PROGRAM MAIN
VAR
	linear_phy_to_adc_test_ 		: linear_phy_to_adc_test;
	linear_adc_to_phy_test_ 		: linear_adc_to_phy_test;
	InterfaceManager_test_ 			: InterfaceManager_test;
	
	coe_handler : CoE_communication_handler;
	interface_manager :InterfaceManager;

	// Terminal_1 : EK1101
	Terminal_2 : EL1808(CoE_communication_handler:=coe_handler );
	Terminal_3 : EL2808(CoE_communication_handler:=coe_handler );
	Terminal_4 : EL4002(CoE_communication_handler:=coe_handler, InterfaceManager:=interface_manager, name:='Terminal_4');
	// Terminal_5 : 
	Terminal_6 : EL3164(CoE_communication_handler:=coe_handler, InterfaceManager:=interface_manager, name:='Terminal_6');
	// Terminal_7 :

END_VAR

TcUnit.RUN();

END_PROGRAM

(* stored: Version 1.1.0.1, ProductVersion 3.1.4024.6
   POU MAIN: Id {040816f1-f230-4b7f-abf9-ea3a3ab6afb7}, SpecialFunc None *)
